(* PLC project motorized_valve, Dassault Systèmes ControlBuild 2024x *)
(* stored: creationDateTime 2023-10-03T11:13:02-01:00 *)

(* This module simulates the behaviour of a motorized valve and its electrical control logic. *)
FUNCTION_BLOCK equipment_library.motorized_valve
  VAR_INPUT
    voltage380 : BOOL := true;
    cmdSupply : BOOL := true;
    sensorSupply : BOOL := true;
  END_VAR
  VAR_INPUT
    openCmd : BOOL := false;
    closeCmd : BOOL := false;
  END_VAR
  VAR_INPUT
    inputFlow : REAL := 0.0;
  END_VAR
  VAR_OUTPUT
    openedSensor : BOOL := false;
    closedSensor : BOOL := false;
    thermal : BOOL := false;
  END_VAR
  VAR_OUTPUT
    openFB : BOOL := false;
    closeFB : BOOL := false;
  END_VAR
  VAR_OUTPUT
    outputFlow : REAL := 0.0;
    percentOpening : REAL := 0.0;
  END_VAR
  VAR
    increment : REAL := 0.0;
    memoOpen : BOOL := false;
    memoClose : BOOL := false;
    openState : BOOL := false;
    closeState : BOOL := false;
    openingVal : REAL := 0.0;
    unit : REAL := 0.0;
  END_VAR
  VAR CONSTANT
    openingTime : REAL := 2.0;
    thermalLogic : BOOL := false;
    openFbLogic : BOOL := true;
    closeFbLogic : BOOL := true;
    openedSensorLogic : BOOL := true;
    closedSensorLogic : BOOL := true;
    flowMax : REAL := 10000.0;
    flowPerHour : BOOL := true;
    flowPerMiinuute : BOOL := false;
  END_VAR
  VAR
    d_locking : BOOL := false;
    v_d_locking : REAL := 0.0;
    d_flow : BOOL := false;
    v_d_flow : REAL := 0.0;
    d_electrical : BOOL := false;
    v_d_electrical : BOOL := false;
    d_closedSensor : BOOL := false;
    v_d_closedSensor : BOOL := false;
    d_openedSensor : BOOL := false;
    v_d_openedSensor : BOOL := false;
    d_closeFB : BOOL := false;
    v_d_closeFB : BOOL := false;
    d_openFB : BOOL := false;
    v_d_openFB : BOOL := false;
  END_VAR


ACTION C_source_code:
/* -----------------------------------------------------------------	*/
/* Type : Model of Operative Behaviour					*/
/* Catégorie :   batch							*/
/* Author : Dassault Systemes						*/
/* Update date : June 2018							*/
/* -----------------------------------------------------------------	*/
/* This module simulates the behaviour of a motorized valve and its 	*/
/* electrical control logic.						*/
/* ----------------------------------------------------------------	*/

/* ----------------------------------------------------------------	*/
/* Management of orders from Control Part					*/
/*	if there is no power supply for command 				*/
/*     the contactors don't understand the control order		*/
/* ----------------------------------------------------------------	*/
if (openCmd && !memoClose && cmdSupply) memoOpen = 1;
if (!openCmd || !cmdSupply) memoOpen = 0;
if (!memoOpen && closeCmd && cmdSupply) memoClose = 1;
if (!closeCmd || !cmdSupply) memoClose = 0;

/* ----------------------------------------------------------------	*/
/* Calculation of the on-state of contactors				*/
/* ----------------------------------------------------------------	*/
openState = memoOpen & voltage380 & ! d_electrical;
closeState = memoClose & voltage380 & ! d_electrical;

/* ----------------------------------------------------------------	*/
/* Management of opening							*/
/* ----------------------------------------------------------------	*/

/* Compute the increment of opening according to the simulation clock*/
increment = CLOCK_PERIOD/1000000;

/* Compute the opening	*/
if (! d_locking) {
	if (openState) {
		openingVal += increment;
		if (openingVal > openingTime)
			openingVal = openingTime;
	}
	if (closeState) {
		openingVal -= increment;
		if (openingVal < 0.0)
			openingVal = 0.0;
	}
}

/* ----------------------------------------------------------------	*/
/* Compute the percentage of opening					*/
/* ----------------------------------------------------------------	*/
if (openingTime > 0.0)
	percentOpening = ((openingVal / openingTime) * 100);

/* ----------------------------------------------------------------	*/
/* Management of flow rate 							*/
/* ----------------------------------------------------------------	*/
if (d_flow)
	outputFlow = v_d_flow;
else {
	outputFlow = percentOpening / 100.0 * inputFlow;
	if (outputFlow > inputFlow) outputFlow = inputFlow;
	if (flowPerHour) unit = 3600.0;
	else if (flowPerMiinuute) unit = 60.0;
		else unit = 1.0;
	if (outputFlow > (flowMax * CLOCK_PERIOD / 1000000)  / unit)
		outputFlow = ((flowMax * CLOCK_PERIOD / 1000000)  / unit) * (percentOpening  /100.0);
}

/* ----------------------------------------------------------------	*/
/* Management of the thermal feedback					*/
/* ----------------------------------------------------------------	*/
if (d_electrical) thermal = v_d_electrical;
else
	thermal = ! thermalLogic && sensorSupply;

/* ----------------------------------------------------------------	*/
/* Management of contatcors' feedback					*/
/* ----------------------------------------------------------------	*/
if (d_openFB) openFB = v_d_openFB;
else
	openFB = (memoOpen ^ ! openFbLogic) && sensorSupply;

if (d_closeFB) closeFB = v_d_closeFB;
else
	closeFB = (memoClose ^ ! closeFbLogic) && sensorSupply;


/* ----------------------------------------------------------------	*/
/* Management of sensors' state						*/
/* ----------------------------------------------------------------	*/
if (d_openedSensor) openedSensor = v_d_openedSensor;
else
	openedSensor = ((openingVal >= openingTime) ^ ! openedSensorLogic) && sensorSupply;

if (d_closedSensor) closedSensor = v_d_closedSensor;
else
	closedSensor = ((openingVal == 0.0) ^ ! closedSensorLogic) && sensorSupply;
END_ACTION
END_FUNCTION_BLOCK
